FUNCTION FC_Check_R : BOOL
VAR_INPUT
	I_sString : REFERENCE TO T_MaxString;
END_VAR
VAR
	stringPos	: INT;
END_VAR

stringPos := FIND(I_sString, 'R');
IF stringPos <> 0 THEN
	I_sString := MID(I_sString, LEN(I_sString), stringPos+1);
	FC_Check_R := TRUE;
ELSE
	FC_Check_R := FALSE;
END_IF

END_FUNCTION

(* stored: Version 1.1.0.1, ProductVersion 3.1.4024.15
   POU FC_Check_R: Id {06715e04-9b73-4b63-b9b5-a8c602534410}, SpecialFunc None *)
